PROGRAM PRG_CML_01_InfeedCtrl
VAR
	tofUnloadInfeedByMETS	: TOF;
	tofInfeedConvDelay		: FB_TOFR;
END_VAR

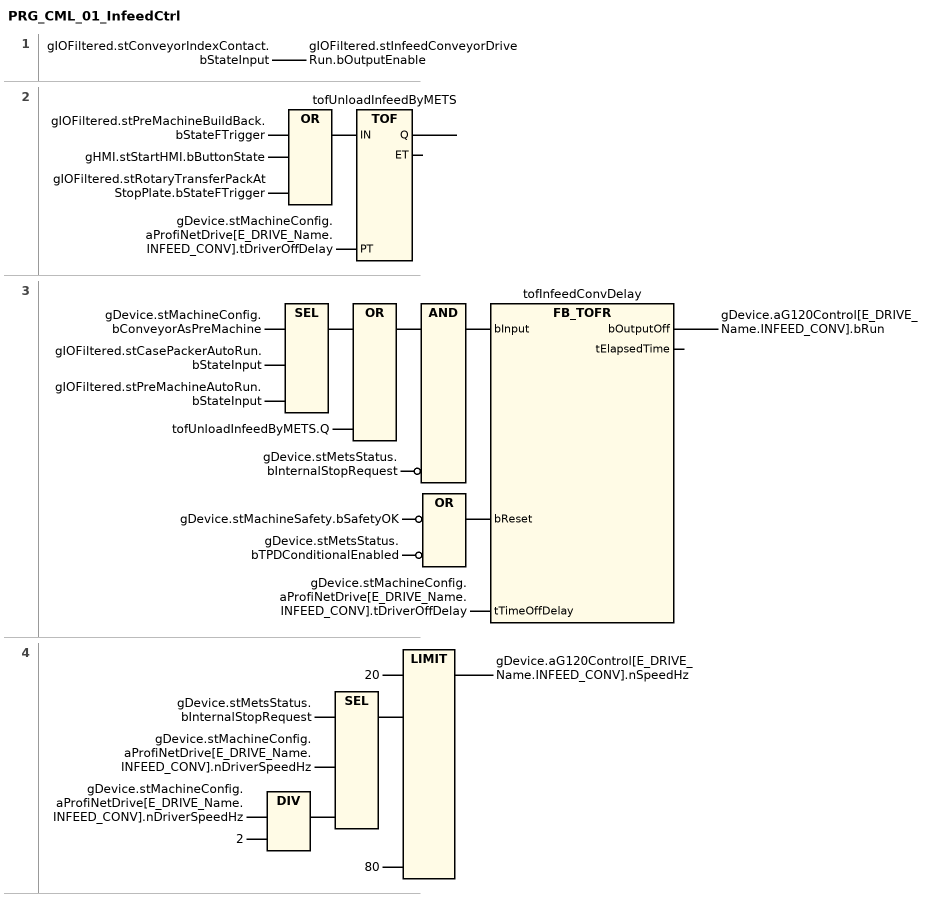
// NETWORK 1
gIOFiltered.stInfeedConveyorDriveRun.bOutputEnable := gIOFiltered.stConveyorIndexContact.bStateInput;

// NETWORK 2
tofUnloadInfeedByMETS(IN := gIOFiltered.stPreMachineBuildBack.bStateFTrigger OR gHMI.stStartHMI.bButtonState OR gIOFiltered.stRotaryTransferPackAtStopPlate.bStateFTrigger, PT := gDevice.stMachineConfig.aProfiNetDrive[E_DRIVE_Name.INFEED_CONV].tDriverOffDelay); // TOF

// NETWORK 3
tofInfeedConvDelay(
    bInput := (SEL(gDevice.stMachineConfig.bConveyorAsPreMachine, gIOFiltered.stCasePackerAutoRun.bStateInput, gIOFiltered.stPreMachineAutoRun.bStateInput) OR tofUnloadInfeedByMETS.Q) AND NOT gDevice.stMetsStatus.bInternalStopRequest,
    bReset := NOT gDevice.stMachineSafety.bSafetyOK OR NOT gDevice.stMetsStatus.bTPDConditionalEnabled,
    tTimeOffDelay := gDevice.stMachineConfig.aProfiNetDrive[E_DRIVE_Name.INFEED_CONV].tDriverOffDelay); // FB_TOFR
gDevice.aG120Control[E_DRIVE_Name.INFEED_CONV].bRun := tofInfeedConvDelay.bOutputOff;

// NETWORK 4
gDevice.aG120Control[E_DRIVE_Name.INFEED_CONV].nSpeedHz := LIMIT(20, SEL(gDevice.stMetsStatus.bInternalStopRequest, gDevice.stMachineConfig.aProfiNetDrive[E_DRIVE_Name.INFEED_CONV].nDriverSpeedHz, gDevice.stMachineConfig.aProfiNetDrive[E_DRIVE_Name.INFEED_CONV].nDriverSpeedHz / 2), 80);

END_PROGRAM

(* stored: Version 1.1.0.1
   POU PRG_CML_01_InfeedCtrl: Id {9bf12203-9051-4b1d-89c6-b97d92677883}, SpecialFunc None *)
